# EPICS IOC start-up script: test/startup/st.mcu024-pils.iocsh
epicsEnvSet("MOTOR_PORT",      "$(SM_MOTOR_PORT=MCU1)")
#epicsEnvSet("IPADDR",          "$(SM_IPADDR=172.30.41.141)")
epicsEnvSet("IPADDR",          "$(SM_IPADDR=127.0.0.1)")
epicsEnvSet("IPPORT",          "$(SM_IPPORT=48898)")
epicsEnvSet("AMSNETIDIOC",     "172.30.38.12.1.1")
epicsEnvSet("ASYN_PORT",       "$(SM_ASYN_PORT=MC_CPU1)")
epicsEnvSet("P",               "$(SM_P=LabS-MCAG:MC-MCU-24:)")
epicsEnvSet("R",               "")
epicsEnvSet("PREC",            "$(SM_PREC=3)")
epicsEnvSet("SM_NOAXES",       "4")
epicsEnvSet("ECM_OPTIONS",     "adsPort=852;amsNetIdRemote=172.30.41.141.1.1;amsNetIdLocal=$(AMSNETIDIOC)"

< ethercatmcController.iocsh

#
# Axis 1
#
epicsEnvSet("AXISCONFIG",      "")
epicsEnvSet("R",               "$(SM_R=m1)")
epicsEnvSet("AXIS_NO",         "$(SM_AXIS_NO=1)")
epicsEnvSet("DESC",            "$(SM_DESC=DESC)")
epicsEnvSet("EGU",             "$(SM_EGU=EGU)")
epicsEnvSet("RAWENCSTEP_ADEL", 0)
epicsEnvSet("RAWENCSTEP_MDEL", 0)
< ethercatmcIndexerAxis.iocsh
< ethercatmcAxisdebug.iocsh

#
# Axis 2
#
epicsEnvSet("AXISCONFIG",      "")
epicsEnvSet("R",               "$(SM_R=m2)")
epicsEnvSet("AXIS_NO",         "$(SM_AXIS_NO=2)")
epicsEnvSet("RAWENCSTEP_ADEL", 0)
epicsEnvSet("RAWENCSTEP_MDEL", 0)
< ethercatmcIndexerAxis.iocsh
< ethercatmcAxisdebug.iocsh

#
# Axis 3
#
epicsEnvSet("AXISCONFIG",      "")
epicsEnvSet("R",               "$(SM_R=m3)")
epicsEnvSet("AXIS_NO",         "$(SM_AXIS_NO=3)")
epicsEnvSet("DESC",            "$(SM_DESC=DESC)")
epicsEnvSet("EGU",             "$(SM_EGU=EGU)")
epicsEnvSet("RAWENCSTEP_ADEL", 0)
epicsEnvSet("RAWENCSTEP_MDEL", 0)
< ethercatmcIndexerAxis.iocsh
< ethercatmcAxisdebug.iocsh

#
# Axis 4
#
epicsEnvSet("AXISCONFIG",      "")
epicsEnvSet("R",               "$(SM_R=m4)")
epicsEnvSet("AXIS_NO",         "$(SM_AXIS_NO=4)")
epicsEnvSet("RAWENCSTEP_ADEL", 0)
epicsEnvSet("RAWENCSTEP_MDEL", 0)
< ethercatmcIndexerAxis.iocsh
< ethercatmcAxisdebug.iocsh

# SoftLimitDelta
epicsEnvSet("R",               "SoftLimitDelta")
epicsEnvSet("CHNO",            "3")
epicsEnvSet("ASYNPARAMNAME",   "SoftLimitDelta")
epicsEnvSet("DESC",            "$(ASYNPARAMNAME)")
epicsEnvSet("PREC",            3)
epicsEnvSet("EGU",             "mm")
< ethercatmcAnalogOutputReadback.iocsh
